// Mitsubishi GX Works2 project: Not_FlibFlob   PLC: Q03UDV

PROGRAM MAIN
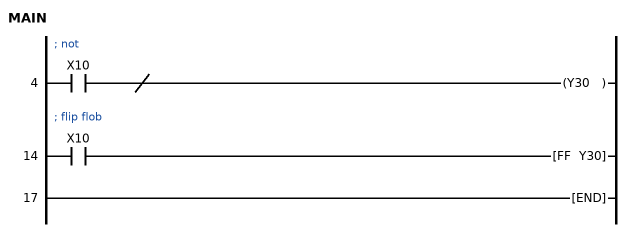
; not
4     LD      X10
      INV
      OUT     Y30
; flip flob
14    LD      X10
      FF      Y30
17    END
END_PROGRAM
